Omron Sysmac Studio project RandNoGen (Sysmac Studio 1.56.0.64011, StandardProject)

# Controller new_Controller_0: NJ501-1500 version 1.64
Units and slaves: Power Supply : NJ-Px3001; CPU : NJ501-1500
Task PrimaryTask (priority 4, period or condition 1000): Program0

VAR_GLOBAL
    Rand_instance : LREAL;
    Random_number : INT;
    A : BOOL := False;
    abc : LREAL;
    numbers : ARRAY[1..10] OF INT;
    k : INT := 1;
    j : INT := 0;
    i : INT := 0;
    B : BOOL := False;
    L : INT := 1;
END_VAR

PROGRAM Program0
VAR
    Rand_instance : Rand;
    RandomG : INT;
    abcd : LREAL;
    Rand_instance2 : Rand;
END_VAR
VAR_EXTERNAL
    Random_number : INT;
    A : BOOL;
    abc : LREAL;
    numbers : ARRAY[1..10] OF INT;
    k : INT;
    j : INT;
    i : INT;
    B : BOOL;
    l : INT;
END_VAR

(* Section Section0: ladder, written here as Structured Text *)

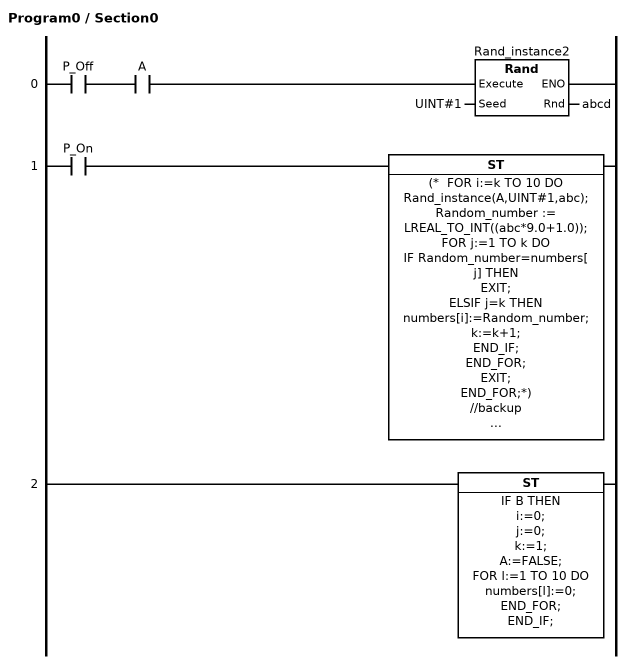
(* Rung 0 *)
Rand_instance2(Execute := P_Off AND A, Seed := UINT#1, Rnd => abcd);
(* Rung 1 *)
IF P_On THEN
    (*	FOR i:=k TO 10 DO
        Rand_instance(A,UINT#1,abc);
        Random_number := LREAL_TO_INT((abc*9.0+1.0));
        FOR j:=1 TO k DO
    
           IF Random_number=numbers[j] THEN
    				EXIT;
    	   ELSIF j=k THEN
    		   numbers[i]:=Random_number;
    		   k:=k+1;
    		END_IF;
        END_FOR;
    			EXIT;
    	END_FOR;*)
    
    //backup
    	FOR i:=k TO 10 DO
        Rand_instance(A,UINT#1,abc);
        Random_number := LREAL_TO_INT((abc*9.0+1.0));
        FOR j:=1 TO 10 DO
    (*        IF Random_number = numbers[j] OR
    			Random_number=0 THEN
    			 j:=j-1;
                EXIT;
    		ELSIF Random_number<>numbers[j] AND 
    				j=i THEN
    				numbers[j] := Random_number;
    				k:=k+1;
    				EXIT;
    		END_IF;*)
           IF Random_number<>numbers[j] AND 
    				j=k THEN
    				numbers[J] := Random_number;
    				k:=k+1;
    				EXIT;
    	   ELSIF Random_number=numbers[j] (*OR numbers[j]=0 *)THEN
    		   EXIT;
    		END_IF;
        END_FOR;
    			EXIT;
    	END_FOR;
    	
    	IF i=11 THEN
    		A:=FALSE;
    	END_IF;
    
    
    
    
    
    (*	FOR i:=k TO 10 DO
        Rand_instance(A,UINT#1,abc);
        Random_number := LREAL_TO_INT((abc*9.0+1.0));
        FOR j:=1 TO k DO
    
           IF Random_number=numbers[j] THEN
    				EXIT;
    	   ELSIF j=k THEN
    		   numbers[i]:=Random_number;
    		   k:=k+1;
    		END_IF;
        END_FOR;
    			EXIT;
    	END_FOR;*)
    	
    	
    (*	FOR i:=k TO 10 DO
        Rand_instance(A,UINT#1,abc);
        Random_number := LREAL_TO_INT((abc*9.0+1.0));
        FOR j:=1 TO k DO
    
           IF j=k THEN
    		   numbers[i]:=Random_number;
    		   k:=k+1;
    	   ELSIF numbers[i]=Random_number THEN
    		   EXIT;
    		END_IF;
        END_FOR;
    			EXIT;
    	END_FOR;*)
    
    
    
    (*	FOR i:=k TO 10 DO
        Rand_instance(A,UINT#1,abc);
        Random_number := LREAL_TO_INT((abc*9.0+1.0));
        FOR j:=1 TO 10 DO
    
           IF Random_number<>numbers[j] AND 
    				j=k THEN
    				numbers[J] := Random_number;
    				k:=k+1;
    				EXIT;
    		END_IF;
        END_FOR;
    			EXIT;
    	END_FOR;*)
    
    (*	FOR i:=1 TO 10 DO
    		IF numbers[i]= 0 THEN
    			numbers[i] := Random_number;
    		END_IF;
    	END_FOR;*)
END_IF;
(* Rung 2 *)
IF B THEN 
		i:=0;
		j:=0;
		k:=1;
		A:=FALSE;
	FOR l:=1 TO 10 DO
		numbers[l]:=0;
	END_FOR;
END_IF;
END_PROGRAM

# Device HMI_NA5_0 (NA): not converted